// TwinCAT 3 PLC project Plc
// ProgramVersion: 3.1.4024.0
// libraries:
//   Tc2_Standard, * (Beckhoff Automation GmbH)
//   Tc2_System, * (Beckhoff Automation GmbH)
//   Tc2_Utilities, * (Beckhoff Automation GmbH)
//   Tc3_Module, * (Beckhoff Automation GmbH)
// project tree:
//   DUTs/ E_Room.TcDUT, ST_Curtain.TcDUT, ST_DigitalLamp.TcDUT, ST_Dimmer.TcDUT, ST_Fan.TcDUT, ST_Room.TcDUT
//   Elements/ Curtain.TcPOU, DigitalLight.TcPOU, Dimmer.TcPOU, Fan.TcPOU
//   GVLs/ GVL.TcGVL, GVL_2.TcGVL
//   / PlcTask.TcTTO
//   POUs/ MAIN.TcPOU, PRG_House.TcPOU, PRG_Testing.TcPOU
//   Rooms/ Bedroom.TcPOU, Hall.TcPOU, Kitchen.TcPOU
//   Utility/ F_Scaling.TcPOU (not stored), RampUp.TcPOU, RampDown.TcPOU
// real-time tasks:
//   TASK PlcTask: cycle T#10ms, priority 20, ADS port 350
//   TASK PlcTask1: cycle T#10ms, priority 21, ADS port 351

CONFIGURATION Plc
    RESOURCE PLC ON TwinCAT3
        TASK PlcTask(INTERVAL := T#10ms, PRIORITY := 20);
        PROGRAM MAIN WITH PlcTask : MAIN;
    END_RESOURCE
END_CONFIGURATION

// ---- DUTs/E_Room.TcDUT
TYPE E_Room :
(
	Hall := 0,
	Kitchen := 1,
	BedRoom1 := 2,
	BedRoom2 := 3
);
END_TYPE

// ---- DUTs/ST_Curtain.TcDUT
TYPE ST_Curtain :
STRUCT
	Open: BOOL;
	Close: BOOL;
	Status: INT;

END_STRUCT
END_TYPE

// ---- DUTs/ST_DigitalLamp.TcDUT
TYPE ST_DigitalLamp :
STRUCT
	PushButton: BOOL;	
	ToggleButton: BOOL;
	Status: BOOL;

END_STRUCT
END_TYPE

// ---- DUTs/ST_Dimmer.TcDUT
TYPE ST_Dimmer :
STRUCT
	DimUp_ON: BOOL;
	DimDown_OFF: BOOL;
	SetBrightness: INT;
	Status: INT;

END_STRUCT
END_TYPE

// ---- DUTs/ST_Fan.TcDUT
TYPE ST_Fan :
STRUCT
	OnOff: BOOL;
	Speed: INT;		//	0: 0%, 1: 25%, 2: 50%, 3: 75%, 4: 100%
	Status: INT;

END_STRUCT
END_TYPE

// ---- DUTs/ST_Room.TcDUT
TYPE ST_Room :
STRUCT
	DigitalLamp	: ARRAY[0..MAX_LAMPS_PER_ROOM] OF ST_DigitalLamp;
	Curtain	: ARRAY[0..MAX_CURTAIN_PER_ROOM] OF ST_Curtain;
	Dimmer	: ARRAY[0..MAX_DIMMER_PER_ROOM] OF ST_Dimmer;
	Fan	: ARRAY[0..MAX_FAN_PER_ROOM] OF ST_Fan;
	Name: STRING;
	
END_STRUCT
END_TYPE

// ---- GVLs/GVL.TcGVL
VAR_GLOBAL
	EL1008_01 AT%I* : ARRAY [0..7] OF BOOL;
	EL1008_02 AT%I* : ARRAY [0..7] OF BOOL;
	EL1008_03 AT%I* : ARRAY [0..7] OF BOOL;
	EL1008_04 AT%I* : ARRAY [0..7] OF BOOL;
	EL1008_05 AT%I* : ARRAY [0..7] OF BOOL;
	EL1008_06 AT%I* : ARRAY [0..7] OF BOOL;
	EL1008_07 AT%I* : ARRAY [0..7] OF BOOL;
	EL1008_08 AT%I* : ARRAY [0..7] OF BOOL;
	
	EL2008_01 AT%Q* : ARRAY [0..7] OF BOOL;
	EL2008_02 AT%Q* : ARRAY [0..7] OF BOOL;
	EL2008_03 AT%Q* : ARRAY [0..7] OF BOOL;
	EL2008_04 AT%Q* : ARRAY [0..7] OF BOOL;
	EL2008_05 AT%Q* : ARRAY [0..7] OF BOOL;
	
	EL4004_01 AT%Q* : ARRAY [0..3] OF INT;
	EL4004_02 AT%Q* : ARRAY [0..3] OF INT;
	EL4004_03 AT%Q* : ARRAY [0..3] OF INT;
	EL4004_04 AT%Q* : ARRAY [0..3] OF INT;
	
	
END_VAR
VAR_GLOBAL CONSTANT
	MAX_ROOM: INT := 3;
	T_LONG_PRESS: TIME := T#2S;
	RAMP_UP_TIME : TIME := T#5S;
	RAMP_DOWN_TIME : TIME := T#5S;
	PLC_CYCLE_TIME_ms : REAL := 10;	
	CURTAIN_OPEN_TIME: TIME := T#5S;
	CURTAIN_CLOSE_TIME: TIME := T#5S;	
	FAN_SPEED_CHANGE_WINDOW: TIME := T#2S;
END_VAR

// ---- GVLs/GVL_2.TcGVL
VAR_GLOBAL
	// Soft inputs (from Application)
	stDeviceControl: ARRAY [0..MAX_ROOM] OF ST_Room := 
	[(Name := 'Hall'), (Name := 'Kitchen'), (Name := 'BedRoom1'), (Name := 'BedRoom2')];
	eRoom : E_Room;
	
END_VAR
VAR_GLOBAL CONSTANT
	
	MAX_LAMPS_PER_ROOM: INT := 4;
	MAX_CURTAIN_PER_ROOM: INT:= 1;
	MAX_DIMMER_PER_ROOM: INT:= 4;
	MAX_FAN_PER_ROOM: INT:= 0;
	
END_VAR

// ---- POUs/MAIN.TcPOU
PROGRAM MAIN
VAR
END_VAR


	PRG_House();
	PRG_Testing();

END_PROGRAM

// ---- POUs/PRG_House.TcPOU
PROGRAM PRG_House
VAR
	hall : Hall;
END_VAR


	hall();
	

////	IO Mapping:
////	Hall:
//	EL1008_01;
//	EL1008_02;
//	EL1008_03;
//	EL2008_01;
//	EL2008_02;
//	EL4004_01;
	
////	Kitchen
//	EL1008_04;
//	EL2008_03;
//	EL4004_02;
	
////	Bedroom1
//	EL1008_05;
//	EL1008_06;
//	EL2008_04;
//	EL4004_03;
	
////	Bedroom2
//	EL1008_07;
//	EL1008_08;
//	EL2008_05;
//	EL4004_04;

END_PROGRAM

// ---- Rooms/Hall.TcPOU
FUNCTION_BLOCK Hall
VAR_INPUT
END_VAR
VAR_OUTPUT
END_VAR
VAR
	lamp01:	DigitalLight;
	lamp02:	DigitalLight;
	lamp03:	DigitalLight;
	dimmer01 : Dimmer;
	curtain: Curtain;
	CurtainMode: INT := 0;
	fan: Fan;
END_VAR


//	IO Mapping - IP

	lamp01.input			:=	EL1008_01[0] OR stDeviceControl[E_Room.Hall].DigitalLamp[0].PushButton;			
	lamp02.input			:=	EL1008_01[1] OR stDeviceControl[E_Room.Hall].DigitalLamp[1].PushButton;			
	lamp03.input			:=	EL1008_01[2] OR stDeviceControl[E_Room.Hall].DigitalLamp[2].ToggleButton;			
	EL1008_01[3];			
	EL1008_01[4];
	EL1008_01[5];
	EL1008_01[6];
	EL1008_01[7];
	
	dimmer01.DimUp_ON		:=	EL1008_02[0] OR stDeviceControl[E_Room.Hall].Dimmer[0].DimUp_ON;
	dimmer01.DimDown_OFF	:=	EL1008_02[1] OR stDeviceControl[E_Room.Hall].Dimmer[0].DimDown_OFF;
	EL1008_02[2];
	EL1008_02[3];
	fan.OnOff				:=	EL1008_02[4] OR stDeviceControl[E_Room.Hall].Fan[0].OnOff;
	fan.speed				:=	EL1008_02[5] (*OR stDeviceControl[E_Room.Hall].Fan[0].Speed*);
	EL1008_02[6];
	EL1008_02[7];

	curtain.openCmd			:=	EL1008_03[0] OR stDeviceControl[E_Room.Hall].Curtain[0].Open;
	curtain.closeCmd		:=	EL1008_03[1] OR stDeviceControl[E_Room.Hall].Curtain[0].Close;
	curtain.IsOpened		:=	EL1008_03[2];
	curtain.IsClosed		:=	EL1008_03[3];
	EL1008_03[4];
	EL1008_03[5];
	EL1008_03[6];
	EL1008_03[7];

//	########################################################################
	
	lamp01(input:=	, keyType:= 0);	
	lamp02(input:=	, keyType:= 0);
	lamp03(input:=	, keyType:= 1);
	
	dimmer01(DimUp_ON:= , DimDown_OFF:= );
	
	curtain(
		openCmd				:= , 
		closeCmd			:= , 
		OpenTime			:= CURTAIN_OPEN_TIME, 
		CloseTime			:= CURTAIN_CLOSE_TIME, 
		IsOpened			:= , 
		IsClosed			:= , 
		mode				:= CurtainMode, 
		open_op				=> , 
		close_op			=> , 
		openClose_perc		=> );

	fan(OnOff:= , speed:= , output=> );

//	########################################################################
//	IO Mapping - OP
	EL2008_01[0]			:=	lamp01.Q;
	EL2008_01[1]			:=	lamp01.Q;
	EL2008_01[2]			:=	lamp02.Q;
	EL2008_01[3]			:=	lamp03.Q;
	EL2008_01[4];
	EL2008_01[5];
	EL2008_01[6];
	EL2008_01[7];

	EL2008_02[0]			:=	curtain.open_op;
	EL2008_02[1]			:=	curtain.close_op;
	EL2008_02[2];
	EL2008_02[3];
	EL2008_02[4];
	EL2008_02[5];
	EL2008_02[6];
	EL2008_02[7];

	EL4004_01[0]			:=	dimmer01.output;
	EL4004_01[1];
	EL4004_01[2];
	EL4004_01[3];

	EL4004_02[0]			:=	fan.output;
	EL4004_02[1];
	EL4004_02[2];
	EL4004_02[3];


//===================================================
EL1008_02[5]	:=	FALSE;


	stDeviceControl[E_Room.Hall].DigitalLamp[0].Status			:=	lamp01.Q;
	stDeviceControl[E_Room.Hall].DigitalLamp[0].Status			:=	lamp01.Q;
	stDeviceControl[E_Room.Hall].DigitalLamp[1].Status			:=	lamp02.Q;
	stDeviceControl[E_Room.Hall].DigitalLamp[2].Status			:=	lamp03.Q;

	stDeviceControl[E_Room.Hall].Curtain[0].Status				:=	0;	//curtain.openClose_perc;
	
	stDeviceControl[E_Room.Hall].Dimmer[0].Status				:=	REAL_TO_INT(F_Scaling(dimmer01.output,0, 32767, 0, 100));
	
	stDeviceControl[E_Room.Hall].Fan[0].Status					:=	REAL_TO_INT(F_Scaling(fan.output,0, 32767, 0, 100));

END_FUNCTION_BLOCK

// ---- Elements/DigitalLight.TcPOU
FUNCTION_BLOCK DigitalLight
VAR_INPUT
	input: BOOL;
	keyType : INT;		//	0: Tap | 1: Toggle
END_VAR
VAR_OUTPUT
	Q : BOOL;
	
END_VAR
VAR
	rtOnOff: R_TRIG;
END_VAR

IF keyType = 0 THEN
	rtOnOff(CLK:= input, Q=> );
	IF rtOnOff.Q THEN
		Q := NOT Q;
	END_IF
ELSIF keyType = 1 THEN
	Q		:=	input;
ELSE
	Q		:=	FALSE;
END_IF

END_FUNCTION_BLOCK

// ---- Elements/Dimmer.TcPOU
FUNCTION_BLOCK Dimmer
VAR_INPUT
	DimUp_ON: BOOL;
	DimDown_OFF: BOOL;
END_VAR
VAR_OUTPUT
	output: INT;
END_VAR
VAR
	tonLongPress_01: TON;
	tonLongPress_02: TON;
	step: INT;
	dimmer_perc: REAL;

	rampUp: RampUp;
	rampDown: RampDown;
END_VAR

	
CASE step OF
	0:	//	Key pressed
		IF DimUp_ON THEN
			step := 10;
		ELSIF DimDown_OFF THEN
			step := 50;	
		END_IF
		rampUp(IN := FALSE, output:= dimmer_perc);
		rampDown(In := FALSE, output:= dimmer_perc);
		tonLongPress_01(IN := FALSE);
		tonLongPress_02(IN := FALSE);
		
		
	10:	//	Short Press - On
		tonLongPress_01(IN:= DimUp_ON, PT:= T_LONG_PRESS, Q=> , ET=> );
		IF tonLongPress_01.Q THEN
			step :=	20;
		ELSIF (NOT DimUp_ON) THEN
			dimmer_perc	:=	32767;
			step		:=	0;
		END_IF
	
	20: // Long Press - Up
		rampUp(
			IN:= TRUE, 
			RampUpTime:= RAMP_UP_TIME, 
			Ramp_lowerLimit:= 0, 
			Ramp_upperLimit:= 32767, 
			output:= dimmer_perc, 
			InProgress=> );
			
		IF (NOT DimUp_ON) THEN
			step	:=	0;
		END_IF
	

	50:	//	Short press - Off
		tonLongPress_02(IN:= DimDown_OFF, PT:= T_LONG_PRESS, Q=> , ET=> );
		IF tonLongPress_02.Q THEN
			step :=	60;
		ELSIF (NOT DimDown_OFF) THEN
			dimmer_perc	:=	0;
			step		:=	0;
		END_IF
	
	60:	//	Long press - Down
		rampDown(
			IN:= TRUE, 
			RampDownTime:= RAMP_DOWN_TIME, 
			Ramp_lowerLimit:= 0, 
			Ramp_upperLimit:= 32767, 
			output:= dimmer_perc, 
			InProgress=> );
		
		IF (NOT DimDown_OFF) THEN
			step	:=	0;
		END_IF
	
END_CASE
	
	output	:=	REAL_TO_INT(dimmer_perc);

END_FUNCTION_BLOCK

// ---- Utility/RampUp.TcPOU
FUNCTION_BLOCK RampUp
VAR_INPUT
	IN: BOOL;
	RampUpTime: TIME;
	Ramp_lowerLimit: REAL;
	Ramp_upperLimit: REAL;
END_VAR
VAR_IN_OUT
	output: REAL;
END_VAR
VAR_OUTPUT
	InProgress: BOOL;	
END_VAR
VAR
	rampUp: REAL;
	x: REAL;
	init: BOOL;
END_VAR


	IF IN THEN
		IF NOT init THEN
			init	:=	TRUE;
			InProgress	:=	TRUE;
			rampUp	:=	TIME_TO_REAL(RampUpTime);		
			x		:=	PLC_CYCLE_TIME_ms / rampUp;
			x		:=	(Ramp_upperLimit - Ramp_lowerLimit) * x;	
		END_IF
		
		IF (output < Ramp_upperLimit) AND (InProgress) THEN
			output		:=	output + x;
		ELSE
			output		:=	Ramp_upperLimit;
			InProgress	:=	FALSE;
		END_IF
		
	ELSE
		InProgress 	:=	FALSE;	
		init		:=	FALSE;
	END_IF

END_FUNCTION_BLOCK

// ---- Utility/RampDown.TcPOU
FUNCTION_BLOCK RampDown
VAR_INPUT
	IN: BOOL;
	RampDownTime: TIME;
	Ramp_lowerLimit: REAL;
	Ramp_upperLimit: REAL;
END_VAR
VAR_IN_OUT
	output: REAL;
END_VAR
VAR_OUTPUT
	InProgress: BOOL;	
END_VAR
VAR
	rampDown: REAL;
	x: REAL;
	init: BOOL;
END_VAR


	IF IN THEN
		IF NOT init THEN
			init	:=	TRUE;
			InProgress	:=	TRUE;
			rampDown	:=	TIME_TO_REAL(RampDownTime);		
			x		:=	PLC_CYCLE_TIME_ms / rampDown;
			x		:=	(Ramp_upperLimit - Ramp_lowerLimit) * x;
		END_IF
		
		IF (output > Ramp_lowerLimit) AND (InProgress) THEN
			output		:=	output - x;
		ELSE
			output		:=	Ramp_lowerLimit;
			InProgress	:=	FALSE;
		END_IF
		
	ELSE
		InProgress 	:=	FALSE;	
		init		:=	FALSE;
	END_IF

END_FUNCTION_BLOCK

// ---- Elements/Curtain.TcPOU
FUNCTION_BLOCK Curtain
VAR_INPUT
	openCmd: BOOL;
	closeCmd: BOOL;
	OpenTime: TIME;
	CloseTime: TIME;
	IsOpened: BOOL;
	IsClosed: BOOL;
	mode: INT;	//	0: keep open/close pressed till fully open/close, release to stop moving 
				//	1: press once, curtain will fully open/close (as per opening time), to stop in between, press any key again
				//	2: curtain with open/close sensor (press once)
END_VAR
VAR_OUTPUT
	open_op: BOOL;
	close_op: BOOL;
	openClose_perc: INT;
END_VAR
VAR
	rampUp: RampUp;
	rampDown: RampDown;
	rtOpenCmd: R_TRIG;
	rtCloseCmd: R_TRIG;
	tofOpen: TOF;
	tofClose: TOF;
	ftOpenCmd: F_TRIG;
	ftCloseCmd: F_TRIG;
END_VAR


	IF mode = 0 THEN
	
		open_op		:=	openCmd AND (NOT closeCmd);
		close_op	:=	closeCmd AND (NOT openCmd);
	
//		rampUp(
//			IN:= (openCmd) AND (NOT closeCmd), 
//			RampUpTime:= OpenTime, 
//			Ramp_lowerLimit:= 0, 
//			Ramp_upperLimit:= 100, 
//			output:= openClose_perc, 
//			InProgress=> open_op);
			
//		rampDown(
//			IN:= (NOT openCmd) AND (closeCmd), 
//			RampDownTime:= CloseTime, 
//			Ramp_lowerLimit:= 0, 
//			Ramp_upperLimit:= 100, 
//			output:= openClose_perc, 
//			InProgress=> close_op);
		
	ELSIF mode = 1 THEN
		rtOpenCmd(CLK:= openCmd, Q=> );
		rtCloseCmd(CLK:= closeCmd, Q=> );
		tofOpen(IN:= rtOpenCmd.Q, PT:= OpenTime, Q=> , ET=> );
		tofClose(IN:= rtCloseCmd.Q, PT:= CloseTime, Q=> , ET=> );
		ftOpenCmd(CLK:= tofOpen.Q, Q=> );
		ftCloseCmd(CLK:= tofClose.Q, Q=> );
		
		IF rtOpenCmd.Q THEN
			open_op		:=	NOT open_op;
		END_IF
		IF ftOpenCmd.Q THEN
			open_op		:=	FALSE;
		END_IF
		
		IF rtCloseCmd.Q THEN
			close_op	:=	NOT close_op;
		END_IF
		IF ftCloseCmd.Q THEN
			close_op	:=	FALSE;
		END_IF
		
	ELSIF mode = 2 THEN
		rtOpenCmd(CLK:= openCmd, Q=> );
		rtCloseCmd(CLK:= closeCmd, Q=> );
		
		IF rtOpenCmd.Q AND (NOT IsOpened) THEN
			open_op		:=	NOT open_op;
		END_IF
		IF IsOpened THEN
			open_op		:=	FALSE;
		END_IF
		
		IF rtCloseCmd.Q AND (NOT IsClosed) THEN
			close_op	:=	NOT close_op;
		END_IF
		IF IsClosed THEN
			close_op	:=	FALSE;
		END_IF
		
	ELSE
		open_op			:=	FALSE;
		close_op		:=	FALSE;
	END_IF

END_FUNCTION_BLOCK

// ---- Elements/Fan.TcPOU
FUNCTION_BLOCK Fan
VAR_INPUT
	OnOff: BOOL;
	speed: BOOL;
	
END_VAR
VAR_OUTPUT
	output: INT;
END_VAR
VAR
	speed_perc: REAL;
	speed_lastNonZeroValue: REAL;
	rtOnOff: R_TRIG;
	rtSpeedChange: R_TRIG;
	step: INT;
	M_OnOff: BOOL;
	tofMonitoringWindow: TOF;
END_VAR


	rtOnOff(CLK:= OnOff, Q=> );
	rtSpeedChange(CLK:= speed, Q=> );
	
	speed_lastNonZeroValue	:=	LIMIT( 25, speed_lastNonZeroValue , 100);
	IF rtOnOff.Q THEN
		IF speed_perc = 0 THEN
			speed_perc		:=	speed_lastNonZeroValue;
			M_OnOff			:=	TRUE;
		ELSE
			speed_perc		:=	0;
			M_OnOff			:=	FALSE;
		END_IF
	END_IF

	CASE step OF
	0:	
		IF rtSpeedChange.Q THEN
			tofMonitoringWindow(IN:= TRUE, PT:= FAN_SPEED_CHANGE_WINDOW, Q=> , ET=> );
			step			:=	10;
		END_IF
		
	10:
		tofMonitoringWindow(IN:= FALSE, PT:= FAN_SPEED_CHANGE_WINDOW, Q=> , ET=> );
		IF tofMonitoringWindow.Q AND rtSpeedChange.Q THEN
			tofMonitoringWindow(IN:= TRUE, PT:= FAN_SPEED_CHANGE_WINDOW, Q=> , ET=> );
			step			:=	20;
		END_IF
		IF NOT tofMonitoringWindow.Q THEN
			speed_perc		:=	25;
			speed_lastNonZeroValue	:=	speed_perc;
			step			:=	0;
		END_IF
		
	20:
		tofMonitoringWindow(IN:= FALSE, PT:= FAN_SPEED_CHANGE_WINDOW, Q=> , ET=> );
		IF tofMonitoringWindow.Q AND rtSpeedChange.Q THEN
			tofMonitoringWindow(IN:= TRUE, PT:= FAN_SPEED_CHANGE_WINDOW, Q=> , ET=> );
			step			:=	30;
		END_IF
		IF NOT tofMonitoringWindow.Q THEN
			speed_perc		:=	50;
			speed_lastNonZeroValue	:=	speed_perc;
			step			:=	0;
		END_IF

	30:
		tofMonitoringWindow(IN:= FALSE, PT:= FAN_SPEED_CHANGE_WINDOW, Q=> , ET=> );
		IF tofMonitoringWindow.Q AND rtSpeedChange.Q THEN
			tofMonitoringWindow(IN:= TRUE, PT:= FAN_SPEED_CHANGE_WINDOW, Q=> , ET=> );
			step			:=	40;
		END_IF
		IF NOT tofMonitoringWindow.Q THEN
			speed_perc		:=	75;
			speed_lastNonZeroValue	:=	speed_perc;
			step			:=	0;
		END_IF
	
	40:
		speed_perc		:=	100;
		speed_lastNonZeroValue	:=	speed_perc;
	
		tofMonitoringWindow(IN:= FALSE, PT:= FAN_SPEED_CHANGE_WINDOW, Q=> , ET=> );
		IF NOT tofMonitoringWindow.Q THEN
			step			:=	0;
		END_IF
		
//		tofMonitoringWindow(IN:= FALSE, PT:= FAN_SPEED_CHANGE_WINDOW, Q=> , ET=> );
//		IF tofMonitoringWindow.Q AND rtSpeedChange.Q THEN
//			tofMonitoringWindow(IN:= TRUE, PT:= FAN_SPEED_CHANGE_WINDOW, Q=> , ET=> );
//			step			:=	0;
//		END_IF
//		IF NOT tofMonitoringWindow.Q THEN
//			speed_perc		:=	100;
//			step			:=	0;
//		END_IF
		
	END_CASE
 	
	tofMonitoringWindow();
	
	output	:=	REAL_TO_INT(F_Scaling(
								Variable_In:= speed_perc, 
								ZeroIn:= 0, 
								ZeroOut:= 100, 
								SpanIn:= 0, 
								SpanOut:= 32767));

END_FUNCTION_BLOCK

// ---- POUs/PRG_Testing.TcPOU
PROGRAM PRG_Testing
VAR
	rampUp: RampUp;
	rampDown: RampDown;
	in: BOOL;
	output: REAL;
	ton1: TON;
	ET: TIME;
	in2: BOOL;
	output2: REAL;
	ton2: TON;
	ET2: TIME;
	openCmd: BOOL;
	closeCmd: BOOL;
	mode: INT;
	open_op: BOOL;
	close_op: BOOL;
	curtain: Curtain;
	openClose_perc: REAL;
	IsOpened: BOOL;
	IsClosed: BOOL;
END_VAR


rampUp(
	IN:= in, 
	RampUpTime:= T#6S345MS, 
	Ramp_lowerLimit:= 100, 
	Ramp_upperLimit:= 700, 
	output:= output, 
	InProgress=> );
	
	ton1(IN:= rampUp.InProgress, PT:= T#1H, Q=> , ET=> );
	IF ton1.IN THEN
		ET	:=	ton1.ET;
	END_IF

rampDown(
	IN:= in2, 
	RampDownTime:= T#6S345MS, 
	Ramp_lowerLimit:= 100, 
	Ramp_upperLimit:= 700, 
	output:= output, 
	InProgress=> );

	ton2(IN:= rampDown.InProgress, PT:= T#1H, Q=> , ET=> );
	IF ton2.IN THEN
		ET2	:=	ton2.ET;
	END_IF	
			
curtain(
	openCmd:= openCmd, 
	closeCmd:= closeCmd, 
	OpenTime:= T#5S, 
	CloseTime:= T#7S, 
	IsOpened:= IsOpened, 
	IsClosed:= IsClosed, 
	mode:= mode, 
	open_op=> open_op, 
	close_op=> close_op,
	openClose_perc=> openClose_perc);

END_PROGRAM

// ---- Rooms/Kitchen.TcPOU
FUNCTION_BLOCK Kitchen
VAR_INPUT
END_VAR
VAR_OUTPUT
END_VAR
VAR
END_VAR

END_FUNCTION_BLOCK

// ---- Rooms/Bedroom.TcPOU
FUNCTION_BLOCK Bedroom
VAR_INPUT
END_VAR
VAR_OUTPUT
END_VAR
VAR
END_VAR

END_FUNCTION_BLOCK
